FUNCTION_BLOCK FB_HSSController_Test EXTENDS FB_TestSuite
VAR
END_VAR

END_FUNCTION_BLOCK

(* stored: Version 1.1.0.1, ProductVersion 3.1.4024.6
   POU FB_HSSController_Test: Id {f5de085e-b521-4344-a831-832f06898f03}, SpecialFunc None *)
